// TIA Portal V17 export
// export: Created 2025-03-07T09:18:26.2445226Z, ExportSetting WithDefaults, DisplayName Totally Integrated Automation Portal, DisplayVersion V17 Update 8, DisplayName TIA Portal Openness, DisplayVersion V17 Update 8, DisplayName TIA Portal Version Control Interface, DisplayVersion V17, DisplayName SINAMICS Startdrive Advanced, DisplayVersion V17 SP2, DisplayName SINAMICS Startdrive G110M, G120, G120C, G120D, G120P, G115D, DisplayVersion V17 SP2, DisplayName SINAMICS Startdrive G130, G150, S120, S150, SINAMICS MV, S210, DisplayVersion V17 SP2, DisplayName STEP 7 Professional, DisplayVersion V17 Update 8, DisplayName SINUMERIK ONE STEP 7 Toolbox, DisplayVersion V17 Update 12, DisplayName SINUMERIK 840D sl STEP 7 Toolbox, DisplayVersion V17 Update 12, DisplayName STEP 7 Safety, DisplayVersion V17 Update 6, DisplayName WinCC Advanced, DisplayVersion V17 Update 8
DATA_BLOCK "DB1802_STA3_CLEANING_VALVE_UNIT_02"   // DB1802
VERSION : 0.1
// stored: AutoNumber false, DBAccessibleFromOPCUA true, DBAccessibleFromWebserver true, InstanceOfName FB1801_STA3_CLEANING_VALVE, InstanceOfType FB
"FB1801_STA3_CLEANING_VALVE"
   // VAR_INPUT
   //    SWITCH_ON_GEN_CON : Bool;
   //    SWITCH_ON_CON : Bool;
   //    SWITCH_ON_AUTO_REQ : Bool;
   //    SWITCH_OFF_CON : Bool;
   //    SWITCH_OFF_AUTO_REQ : Bool;
   //    HMI_LINE_REQ : Bool;
   //    UNIT_ALARM : UInt;
   //    STATION_ALARM : UInt;
   // END_VAR
   // VAR_OUTPUT
   //    SWITCHED_ON : Bool;
   //    SWITCHED_OFF : Bool;
   //    HMI_MOTION_EXECUTABILITY_LEFT : Bool;
   //    HMI_MOTION_EXECUTABILITY_RIGHT : Bool;
   //    HMI_MOTION_END_POS_LEFT : Bool;
   //    HMI_MOTION_END_POS_RIGHT : Bool;
   //    SWITCH_ON : Bool;
   //    SWITCH_OFF : Bool;
   // END_VAR
   // VAR
   //    VALVE : "ASPIRATION";
   // END_VAR
   // VAR RETAIN
   //    TIMER_SIMULTANEITY { S7_SetPoint := 'True'} : TON_TIME;
   //    TIMER_TIME_EXCEEDED { S7_SetPoint := 'True'} : TON_TIME;
   // END_VAR
BEGIN
END_DATA_BLOCK
